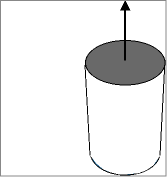
VISUALIZATION VISU_Tube_Top_7  // 167x177
VAR_IN_OUT
	azi : LREAL;
END_VAR
    Ellipse (90,130 70x45)
        p2858320360: azi
    Polygon (85,60) (165,60) (160,155) (153,165) (146,170) (138,173) (127,174) (118,174) (110,172) (103,169) (96,163) (90,155)
        p2858320360: azi
    Ellipse (85,40 80x45)
        p2858320360: azi
    Polygon (120,10) (125,0) (130,10)
        p2858320360: azi
    Polyline (125,60) (125,10)
        p2858320360: azi
    Polyline (160,155) (165,60)
        p2858320360: azi
    Polyline (90,155) (85,65)
        p2858320360: azi
END_VISUALIZATION

(* stored: Version 1.1.0.1, ProductVersion 3.1.4018.5
   Visu VISU_Tube_Top_7: Id {677398bc-927e-437e-b489-ef5a7c3cf0bd} *)
